Staubli VAL3: splitWord.pgx

public program splitWord(string& x_sInput[], lists& x_lResult[])
  local num l_nLength
  local num l_nElement
  local string l_sLine
  local num l_nCount
begin

  l_nLength = size(x_sInput)
  resize(x_lResult,1,1)
  resize(x_lResult.sString,1,1)
  x_lResult.sString =""
  resize(x_lResult,1,l_nLength)

  // iterate complete input x_sInput[0] ... x_sInput[l_nLength-1]
  for l_nElement = 0 to l_nLength-1

    // copy element
    l_sLine = x_sInput[l_nElement]

    // search x_sPattern
    l_nCount = 0
    while len(l_sLine)!=0

      if l_nCount != 0
        append(x_lResult[l_nElement].sString)
      endIf

      x_lResult[l_nElement].sString[l_nCount] = left(l_sLine,1)
      l_sLine = right(l_sLine,len(l_sLine)-1)
      l_nCount = l_nCount+1

    endWhile
  endFor


end
